// TIA Portal V17 export
TagTable "Codex_Popup_Sim_Int_Tags"
  Sim_SelectedCompID : Int  (1 s, start 1)   // Selected component ID. 1=Valve01, 2=Heater01, 3=Fan01.
  Sim_ClickPulse : Int  (1 s, start 0)   // Component click trigger pulse.
  Sim_DoubleClickTime_ms : Int  (1 s, start 800)   // Double-click time in milliseconds.
  Sim_Switch1 : Int  (1 s, start 0)   // Simulated Switch[1].
  Sim_RealValue1_Int : Int  (1 s, start 0)   // Integer placeholder for RealValue[1] simulation.
  Sim_Visible : Int  (1 s, start 0)   // Popup visible state.
  Sim_ActiveID : Int  (1 s, start 0)   // Current active popup ID.
  Sim_Confirmed : Int  (1 s, start 0)   // Confirmed state.
  Sim_ConfirmPulse : Int  (1 s, start 0)   // Confirm button pulse.
  Sim_CancelPulse : Int  (1 s, start 0)   // Cancel button pulse.
